// TIA Portal V18 export
DATA_BLOCK "Volume counter"   // DB206
{ S7_Optimized_Access := 'TRUE' }
VERSION : 0.1
// stored: AutoNumber true, DBAccessibleFromOPCUA true, IsOnlyStoredInLoadMemory false, IsRetainMemResEnabled false, IsWriteProtectedInAS false, MemoryReserve 100
   VAR RETAIN
      "A" : Struct
         Impulse : Real := 0.0;
         "Impulse in HMI" : Real := 0.00625;
         "Maximum Down time" : Int;
         "Maximum Down time in sec" : DInt;
         "serial number" : String;
         "Leakage Pulses" : Int;
         "Leakage Control time" : Int;
         "Leakage control time in Sec" : DInt;
      END_STRUCT;
      "B" : Struct
         Impulse : Real;
         "Impulse in HMI" : Real := 0.00625;
         "Maximum Down time" : Int;
         "Maximum Down time in sec" : DInt;
         "serial number" : String;
         "Leakage Pulses" : Int;
         "Leakage Control time" : Int;
         "Leakage control time in Sec" : DInt;
      END_STRUCT;
   END_VAR
   VAR
      "Control A" : Struct
         "Create CV during Process" : Bool;
         "New CV during Process" : DInt;
         "Current Pulses during process" : DInt;
         "Create New CV For ratio check" : Bool;
         "New CV  For ratio check" : DInt;
         "Current Pulses  For ratio check" : DInt;
      END_STRUCT;
      "Control B" : Struct
         "Create CV during Process" : Bool;
         "New CV during Process" : DInt;
         "Current Pulses during process" : DInt;
         "Create New CV For ratio check" : Bool;
         "New CV For ratio check" : DInt;
         "Current Pulses For ratio check" : DInt;
      END_STRUCT;
      "Volume A" : Struct
         "volume For Ratio check" : Real;
         "volume For Qty Display" : Real;
      END_STRUCT;
      "Volume B" : Struct
         "volume For Ratio check" : Real;
         "volume For Qty Display" : Real;
      END_STRUCT;
      Volume : Struct
         "For Process" : Real;
         "For Ratio Check" : Real;
      END_STRUCT;
      "Process running start volume measurement" : Bool;
      "Process running start volume measurement ONS" : Bool;
   END_VAR
   VAR RETAIN
      Selection : Struct
         "A" : Int := 0;
         "B" : Int := 0;
      END_STRUCT;
      Enabled : Struct
         "A" : Bool;
         "B" : Bool;
         AB : Bool;
      END_STRUCT;
   END_VAR
   VAR
      "No signal" : Struct
         "A" : Bool;
         "B" : Bool;
      END_STRUCT;
      "Leakage Control A" : Struct
         "Start Test" : Bool;
         "Start Test ONS" : Bool;
         "New Cv" : DInt;
         pulses : DInt;
         "Reset timer" : Bool;
         F_trigger : Bool;
      END_STRUCT;
      "Leakage Control B" : Struct
         "Start Test" : Bool;
         "Start Test ONS" : Bool;
         "New Cv" : DInt;
         pulses : DInt;
         "Reset timer" : Bool;
         F_trigger : Bool;
      END_STRUCT;
      "Pump leakage" : Struct
         "A" : Bool;
         "B" : Bool;
      END_STRUCT;
   END_VAR
   VAR RETAIN
      "Volume Counter Enable button" : Bool;
   END_VAR
BEGIN
END_DATA_BLOCK
